FUNCTION_BLOCK PICKER_HMI_ADP_NEW (* Composite FB For HMI Plug *)
  (* Standard: 61499-2 *)
  (* Version 0.2, 2003-12-05, JHC, Rockwell Automation, Renamed from NEWCOMPFB. *)
  (* Version 0.1, 2002-01-08, JHC, Rockwell Automation, Added DLY FB as example. *)
  (* Version 0.0, 2000-05-27, JHC, Rockwell Automation *)
  (* Compiler header: package fb.rt.pnp; *)
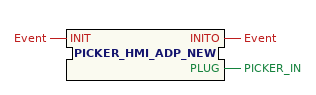
  EVENT_INPUT
    INIT; (* Initialization Request *)
  END_EVENT
  EVENT_OUTPUT
    INITO; (* Initialization Confirm *)
  END_EVENT
  PLUGS
    PLUG : PICKER_IN;
  END_PLUGS
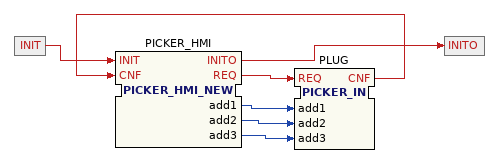
  FBS
    PICKER_HMI : PICKER_HMI_NEW;
  END_FBS
  EVENT_CONNECTIONS
    INIT TO PICKER_HMI.INIT;
    PICKER_HMI.INITO TO INITO;
    PICKER_HMI.REQ TO PLUG.REQ;
    PLUG.CNF TO PICKER_HMI.CNF;
  END_CONNECTIONS
  DATA_CONNECTIONS
    PICKER_HMI.add1 TO PLUG.add1;
    PICKER_HMI.add2 TO PLUG.add2;
    PICKER_HMI.add3 TO PLUG.add3;
  END_CONNECTIONS
END_FUNCTION_BLOCK
